// TIA Portal V16 export
// export: Created 2021-04-11T09:51:28.2546355Z, ExportSetting WithDefaults, DisplayName Totally Integrated Automation Portal, DisplayVersion V16, DisplayName TIA Portal Version Control Interface, DisplayVersion V16, DisplayName TIA Portal Openness, DisplayVersion V16, DisplayName STEP 7 Professional, DisplayVersion V16, DisplayName STEP 7 Safety, DisplayVersion V16, DisplayName WinCC Unified SCADA Engineering System, DisplayVersion V16
DATA_BLOCK "signalKVSStation"   // DB20
{ S7_Optimized_Access := 'TRUE' }
VERSION : 0.1
// stored: AutoNumber false, DBAccessibleFromOPCUA true, IsOnlyStoredInLoadMemory false, IsRetainMemResEnabled false, IsWriteProtectedInAS false, MemoryReserve 100
   VAR
      isWorkControlCircuit : Bool;   // цепи управления активированы
      isStopAlarm : Bool;   // приход любой аварии которая останавливает установку
      isOtherAlarm : Bool;   // приход просто аварий
      isStartAutoMode : Bool;   // начало работы в автоматическом режиме
      enableAutoMode : Bool;   // разрешение перевода в автоматический режим
      isPreparationAutoModeFinish : Bool;   // подготовк к запуску автоматического режима
      enableManualMode : Bool;   // разрешение работы в ручном режиме
      qManualMode : "mode";   // активация катушек в ручном режиме
      qAutoMode : "mode";   // активация катушек в автоматическом режиме
      currentWeight : Array[0..12] of Real;   // вес получаемый по модбасу
      stableWeight : Array[0..12] of "stableWeight";   // установившийся вес в бункерах
   END_VAR
BEGIN
END_DATA_BLOCK
